// TwinCAT 3 PLC project SPS
// ProgramVersion: 3.1.4026.22
// libraries:
//   VisuElemMeter, * (System)
//   VisuElems, * (System)
//   VisuElemsSpecialControls, * (System)
//   VisuElemsWinControls, * (System)
//   VisuElemTextEditor, * (System)
//   VisuInputs, * (System)
//   VisuNativeControl, * (System)
//   Tc2_MC2, * (Beckhoff Automation GmbH)
//   Tc2_Standard, * (Beckhoff Automation GmbH)
//   Tc2_System, * (Beckhoff Automation GmbH)
//   Tc3_IotBase, * (Beckhoff Automation GmbH)
//   VisuSymbols, * (System)
// project tree:
//   GVLs/ GVL_PosKinematic.TcGVL, IFC_HW.TcGVL
//   / PlcTask.TcTTO
//   POUs/Abfüllmodul/ FB_Abfuellmodul.TcPOU, FB_Dispenser.TcPOU, FB_EZylinder.TcPOU, FB_Vereinzelung.TcPOU
//   POUs/ eBetriebszustand.TcDUT, FUN_Scale.TcPOU, MAIN.TcPOU
//   POUs/IoT/ FB_MQTT.TcPOU
//   POUs/Manipulator/ FB_Manipulator.TcPOU
//   POUs/Manipulator/Roboter/ FB_Roboter.TcPOU (not stored), FB_Roboter_Axis.TcPOU (not stored), FB_Roboter_E.TcPOU (not stored), FB_Roboter_Logik.TcPOU (not stored)
//   POUs/Statusleuchte/ FB_Ampelleuchte.TcPOU, FB_Blinklicht.TcPOU
// (motion and I/O tree: see PLC project lf_system_plc)
// real-time tasks:
//   TASK PlcTask: cycle T#10ms, priority 21, ADS port 350
//   TASK PlcTask1: cycle T#10ms, priority 22, ADS port 351
//   TASK PlcTask2: cycle T#10ms, priority 20, ADS port 352
//   TASK PlcTask3: cycle T#10ms, priority 23, ADS port 353
// variable links:

CONFIGURATION SPS
    RESOURCE PLC ON TwinCAT3
        TASK PlcTask(INTERVAL := T#10ms, PRIORITY := 23);
        PROGRAM MAIN WITH PlcTask : MAIN;
    END_RESOURCE
END_CONFIGURATION

// ---- POUs/eBetriebszustand.TcDUT
{attribute 'qualified_only'}
{attribute 'strict'}
{attribute 'to_string'}
TYPE eBetriebszustand :
(
	Off        := 0,   // nicht betriebsbereit
	Error      := 1,   // Fehlerbehafteter Stop
	Setup      := 2,   // Wartung
	Warning    := 3,   // nicht fehlerbehafteter, nicht geplanter Stop
	Init       := 4,   // Herstellung Betriebsbereitschaft
	Ready      := 5,   // betriebsbereit
	Production := 6,   // Betrieb
	Done       := 7,   // Betrieb abgeschlossen
	Stop       := 8
);
END_TYPE

// ---- GVLs/GVL_PosKinematic.TcGVL
{attribute 'qualified_only'}
VAR_GLOBAL
	// Home position
	pXhome : REAL := 29;
	pYhome : REAL := 145.5;
	pZhome : REAL := 45;
	
	// Conveyor position
	pXconv : REAL := 29;
	pYconv : REAL := 145.5;
	pZconv : REAL := 130;
	
	//Scale position
	pXscale : REAL := 36;
	pYscale : REAL := 7.5;
	pZscale : REAL := 131.5;
	
	// Heating position
	pXheat : REAL := 218.5;
	pYheat : REAL := 7;
	pZheat : REAL := 159;
	
	// Storage position
	pX1stor : REAL := 107;
	pX2stor : REAL := 158.7;
	pX3stor : REAL := 209.3;
	pX4stor : REAL := 260.3;
	pYstor : REAL := 139;
	pZstor : REAL := 120;
	
	// Z offset height
	pZoff : REAL := 45;
END_VAR

// ---- GVLs/IFC_HW.TcGVL
// In dieser GVL werden alle Variablen deklariert die auf die realen Klemmen zugreifen
VAR_GLOBAL
	
	// Allgemeine Variablen fur MAIN und HMI
		bEnable		AT%I*	: BOOL;			// Enable Factory (HMI Production Umgebung)
		bExecute	AT%I*	: BOOL;			// Startsignal	(Start Knopf Konsole)
		bStop				: BOOL;			// Stop Variable (interne Variable um FB's zu stoppen)
		
	// Station Statusampel	
		bAmpelRot 	AT%Q* 	: BOOL;			// Signal-LED Rot
		bAmpelGelb 	AT%Q* 	: BOOL;			// Signal-LED Gelb
		bAmpelGrun 	AT%Q* 	: BOOL;			// Signal-LED Grun
			
	// Station Vereinzelung
		bEinzelSens1 	AT%I*	: BOOL;					// Separation Sensor 1 (Kammer)
		bEinzelSens2 	AT%I*	: BOOL;					// Separation Sensor 2 (Rohr)
		bEinzelSens3 	AT%I*	: BOOL;					// Separation Sensor 3 (Flasche auf Kopf)
		bR1AKT1 		AT%Q* 	: BOOL := FALSE;		// Relais 1 Aktor 1 (Schleuse Oben öffnen)
		bR2AKT1 		AT%Q* 	: BOOL := TRUE; 		// Relais 2 Aktor 1 (Schleuse Oben schließen)
		bR1AKT2 		AT%Q* 	: BOOL := FALSE;		// Relais 1 Aktor 2 (Schleuse Unten öffne)
		bR2AKT2 		AT%Q* 	: BOOL := TRUE;			// Relais 2 Aktor 2	(Schleuse Unten schließen)
	
	// Station Forderband
		bBandSens1 	AT %I*	: BOOL;		// Forderband Sensor 1 (Extruder 1)
		bBandSens2	AT %I*	: BOOL;		// Forderband Sensor 2 (Extruder 2)
		bBandSens3 	AT %I*	: BOOL;		// Forderband Sensor 3 (Extruder 3)
		bBandSens4 	AT %I*	: BOOL;		// Forderband Sensor 4 (Übergabe Roboter)
		bBandHub1 	AT %Q*	: BOOL;		// Forderband Hubmagnet 1 (Schleuse Extruder 1)
		bBandHub2 	AT %Q*	: BOOL;		// Forderband Hubmagnet 1 (Schleuse Extruder 2)
		bBandHub3 	AT %Q*	: BOOL;		// Forderband Hubmagnet 1 (Schleuse Extruder 3)
		
		ax_Extruder1 	: AXIS_REF;		// Forderband NC-Achse Extruder 1
		ax_Extruder2 	: AXIS_REF;		// Forderband NC-Achse Extruder 2
		ax_Extruder3 	: AXIS_REF;		// Forderband NC-Achse Extruder 3
		ax_BandMotor 	: AXIS_REF;		// Forderband NC-Achse Band
		
		iBandFullmenge1		: INT := 1;	// in Gramm (Soll Füllmenge Extruder 1)
		iBandFullmenge2		: INT := 1;	// in Gramm (Soll Füllmenge Extruder 2)
		iBandFullmenge3		: INT := 1;	// in Gramm (Soll Füllmenge Extruder 3)
		
	//Füllstandsüberwachung
		iFillSens1 AT%I*	: UINT;		// Füllstandssensor im Granulatspeicher 1
		iFillSens2 AT%I*	: UINT;		// Füllstandssensor im Granulatspeicher 2
		iFillSens3 AT%I*	: UINT;		// Füllstandssensor im Granulatspeicher 3
		
		rFillLevelPercent1	: REAL;		// Füllstand im Granulatspeicher 1 in %
		rFillLevelGramm1	: REAL;		// Füllstand im Granulatspeicher 1 in g
		rFillLevelPercent2	: REAL;		// Füllstand im Granulatspeicher 2 in %
		rFillLevelGramm2	: REAL;		// Füllstand im Granulatspeicher 2 in g
		rFillLevelPercent3	: REAL;		// Füllstand im Granulatspeicher 3 in %
		rFillLevelGramm3	: REAL;		// Füllstand im Granulatspeicher 3 in g
		
		rMaxFillLevel 		: REAL := 375;	// Kalibrierter Füllstand für 10% * 10
		
	// Station Waage
		sWaageNachricht		: STRING;	// Nachricht von Wagezelle (fur virtuelle Inbetriebnahme notig)
		bWaageNull			: BOOL;		// TARA Waage (Waage auf Null setzen)
		iWaageMesswert		: INT;		// Messwert der Waage
		
	// Station Behalteridentifikation
		bIdSensorTrager		: BOOL;		// Sensor bei Erkennung eines Datentrager
		sIdNachricht		: STRING;	// Nachricht von RFID-System (fur virtuelle Inbetriebnahme notig)
		sSeriennummer		: STRING;	// Seriennummer RFID-Tag
		
	//Temperierstation
		bVentilator1 	AT %Q*	: BOOL;		// Ventilator 1
		bVentilator2 	AT %Q*	: BOOL;		// Ventilator 2
		bVentilator3 	AT %Q*	: BOOL;		// Ventilator 3
		
		iTempSens1 		AT%I*	: UINT;		// Temperatursensor 1
		iTempSens2 		AT%I*	: UINT;		// Temperatursensor 2
		iHeizpatrone 	AT%Q*	: UINT;		// Heizpatronen
		
		iMaxTemp				: UINT := 5500;		// in °C * 100
		
	// Station Manipulator
		bManEndXmin 		AT%I* 	: BOOL := TRUE;		// Manipulator min Endschalter Achse x
		bManEndYmin 		AT%I* 	: BOOL := TRUE;		// Manipulator min Endschalter Achse y
		bManEndZmin 		AT%I* 	: BOOL := TRUE;		// Manipulator min Endschalter Achse z
		bManEndGmin 		AT%I* 	: BOOL := TRUE;		// Manipulator min Endschalter Achse Gripper
		bManEndXmax 		AT%I* 	: BOOL := TRUE;		// Manipulator max Endschalter Achse x
		bManEndYmax 		AT%I* 	: BOOL := TRUE;		// Manipulator max Endschalter Achse y
		bManEndZmax 		AT%I* 	: BOOL := TRUE;		// Manipulator max Endschalter Achse z
		bManEndGmax 		AT%I* 	: BOOL := TRUE;		// Manipulator max Endschalter Achse Gripper
		bManBrakeZ			AT%Q*	: BOOL := FALSE;	// Bremse Achse z
		
		ax_ManX			: AXIS_REF;			// Manipulator NC-Achse x
		ax_ManY			: AXIS_REF;			// Manipulator NC-Achse y
		ax_ManZ			: AXIS_REF;			// Manipulator NC-Achse z
		ax_ManG			: AXIS_REF; 		// Manipulator NC-Achse Gripper
		
		bGripperClosed		AT%Q*	: BOOL; 			// signal if gripper is closed ONLY USED IN SIM
END_VAR

// ---- POUs/MAIN.TcPOU
PROGRAM MAIN
VAR
	fb_Ampelleuchte :FB_Ampelleuchte;	
	fb_Abfuellmodul :FB_Abfuellmodul;
	fb_Manipulator :FB_Manipulator;
	
	nState :INT :=0;
	
	fb_MQTT :FB_MQTT;
END_VAR

	
fb_Ampelleuchte(eState:= , bAmpelGruen_out=> IFC_HW.bAmpelGrun, bAmpelRot_out=> IFC_HW.bAmpelRot, bAmpelGelb_out=> IFC_HW.bAmpelGelb);

fb_Abfuellmodul(bEnable:= , bExecute:= , eState=> ); 
fb_Manipulator(bEnable:= , bExecute:= , bGripperClosed=> IFC_HW.bGripperClosed, eState=> );

IF fb_Abfuellmodul.eState = eBetriebszustand.Init OR fb_Manipulator.eState = eBetriebszustand.Init THEN
	fb_Ampelleuchte.eState := eBetriebszustand.init;
ELSIF fb_Abfuellmodul.eState = eBetriebszustand.ready AND fb_Manipulator.eState = eBetriebszustand.ready THEN
	fb_Ampelleuchte.eState := eBetriebszustand.ready;
ELSIF fb_Abfuellmodul.eState = eBetriebszustand.production OR fb_Manipulator.eState = eBetriebszustand.Production THEN
	fb_Ampelleuchte.eState := eBetriebszustand.Production;
ELSIF fb_Abfuellmodul.eState = eBetriebszustand.off AND fb_Manipulator.eState = eBetriebszustand.off THEN
	fb_Ampelleuchte.eState := eBetriebszustand.off;
ELSE 
	fb_Ampelleuchte.eState := eBetriebszustand.Warning;
END_IF


IF NOT IFC_HW.bEnable THEN
	nState :=0;
END_IF
CASE nState Of
	0://off
	fb_Abfuellmodul.bEnable :=FALSE;
	fb_Manipulator.bEnable :=FALSE;
	
	IF IFC_HW.bEnable THEN
		nstate:=1;
	END_IF
	
	1: //init
	fb_Abfuellmodul.bEnable :=TRUE;
	fb_Manipulator.bEnable :=TRUE;
	
	IF fb_Abfuellmodul.eState = eBetriebszustand.Ready AND fb_Manipulator.eState = eBetriebszustand.Ready THEN
		nState:=2;
	END_IF
	
	2: //ready
	IF IFC_HW.bExecute AND iFC_HW.bEinzelSens1 THEN
		nstate :=21;
	END_IF
	IF NOT iFC_HW.bEinzelSens2 AND NOT iFC_HW.bEinzelSens1 THEN
		fb_Abfuellmodul.bEnable :=FALSE;
		nState :=1;
	END_IF
	
	21: //bottle
	fb_Abfuellmodul.bExecute :=TRUE;
	
	IF fb_Abfuellmodul.eState = eBetriebszustand.Done THEN
		fb_Abfuellmodul.bExecute :=FALSE;
		nstate :=22;
	END_IF
	
	22: //mani
	fb_Manipulator.bExecute :=TRUE;
	
	IF fb_Manipulator.eState = eBetriebszustand.Done THEN
		fb_Manipulator.bExecute :=FALSE;
		nState :=23;
	END_IF
	
	23://done
	IF NOT IFC_HW.bExecute THEN
		nState:=2;
	END_IF
END_CASE


fb_MQTT(data:= IFC_HW.bEnable);

END_PROGRAM

// ---- POUs/Statusleuchte/FB_Ampelleuchte.TcPOU
FUNCTION_BLOCK FB_Ampelleuchte
VAR_INPUT
	eState : eBetriebszustand;
END_VAR
VAR_OUTPUT

	
	bAmpelGruen_out :BOOL;
	bAmpelRot_out :BOOL;
	bAmpelGelb_out :BOOL;
	
END_VAR
VAR
	fb_BlinklichtGr :FB_Blinklicht;
	fb_BlinklichtRt :FB_Blinklicht;
	fb_BlinklichtGb :FB_Blinklicht;
	AmpelGruenblinken:BOOL;
	AmpelRotblinken :BOOL;
	AmpelGelbblinken :BOOL;
	bAmpelGruen :BOOL;
	bAmpelRot :BOOL;
	bAmpelGelb :BOOL;
END_VAR

CASE eState OF
	0: //OFF nicht Betriebsbereit
	//keine Lampe leuchtet
	bAmpelGruen :=FALSE;
	bAmpelRot :=FALSE;
	bAmpelGelb :=FALSE;
	AmpelGruenblinken:=FALSE;
	AmpelRotblinken :=FALSE;
	AmpelGelbblinken :=FALSE;
	
	1: //Error Fehlerbehafteter Stop (Sicherheitssteuerung)
	//Rote Lampe Leuchtet 
	bAmpelGruen :=FALSE;
	bAmpelRot :=TRUE;
	bAmpelGelb :=FALSE;
	AmpelGruenblinken:=FALSE;
	AmpelRotblinken :=FALSE;
	AmpelGelbblinken :=FALSE;
	
	2: //Setup Wartung
	//Rot und Gelb blinkt
	bAmpelGruen :=FALSE;
	bAmpelRot :=FALSE;
	bAmpelGelb :=FALSE;
	AmpelGruenblinken:=FALSE;
	AmpelRotblinken :=TRUE;
	AmpelGelbblinken :=TRUE;
	
	3: //Warning Nicht Fehlerbehafteter nicht geplanter Stop
	//Gelb blinken
	bAmpelGruen :=FALSE;
	bAmpelRot :=FALSE;
	bAmpelGelb :=FALSE;
	AmpelGruenblinken:=FALSE;
	AmpelRotblinken :=FALSE;
	AmpelGelbblinken :=TRUE;
	
	4: //Init Herstellung Betriebsbereitschaft
	//Gelb Grün blinkt
	bAmpelGruen :=FALSE;
	bAmpelRot :=FALSE;
	bAmpelGelb :=FALSE;
	AmpelGruenblinken:=TRUE;
	AmpelRotblinken :=FALSE;
	AmpelGelbblinken :=TRUE;
	
	5: //Ready Betriebsbereit
	//Grün blinkt
	bAmpelGruen :=FALSE;
	bAmpelRot :=FALSE;
	bAmpelGelb :=FALSE;
	AmpelGruenblinken:=TRUE;
	AmpelRotblinken :=FALSE;
	AmpelGelbblinken :=FALSE;
	
	6: //Production Betrieb
	//Grün leuchtet
	bAmpelGruen :=TRUE;
	bAmpelRot :=FALSE;
	bAmpelGelb :=FALSE;
	AmpelGruenblinken:=FALSE;
	AmpelRotblinken :=FALSE;
	AmpelGelbblinken :=FALSE;
	
	7: //Done Betrieb abgeschlossen 
	//Grün Gelb leuchten
	bAmpelGruen :=TRUE;
	bAmpelRot :=FALSE;
	bAmpelGelb :=TRUE;
	AmpelGruenblinken:=FALSE;
	AmpelRotblinken :=FALSE;
	AmpelGelbblinken :=FALSE;
	
	8: //Stop
	//Rot blinken
	bAmpelGruen :=FALSE;
	bAmpelRot :=FALSE;
	bAmpelGelb :=FALSE;
	AmpelGruenblinken:=FALSE;
	AmpelRotblinken :=TRUE;
	AmpelGelbblinken :=FALSE;
END_CASE

fb_BlinklichtGb(bStartStop:= AmpelGelbblinken, tPeriod:= T#1S , bBlink=> );
fb_BlinklichtGr(bStartStop:= AmpelGruenblinken, tPeriod:= T#1S, bBlink=> );
fb_BlinklichtRt(bStartStop:= AmpelRotblinken, tPeriod:= T#1S, bBlink=> );

IF fb_BlinklichtGb.bBlink OR bAmpelGelb THEN
	bAmpelGelb_out :=TRUE;
ELSE
	bAmpelGelb_out :=FALSE;
END_IF
IF fb_BlinklichtGr.bBlink OR bAmpelGruen THEN
	bAmpelGruen_out :=TRUE;
ELSE
	bAmpelGruen_out :=FALSE;
END_IF
IF fb_BlinklichtRt.bBlink OR bAmpelRot THEN
	bAmpelRot_out :=TRUE;
ELSE
	bAmpelRot_out :=FALSE;
END_IF

END_FUNCTION_BLOCK

// ---- POUs/Statusleuchte/FB_Blinklicht.TcPOU
FUNCTION_BLOCK FB_Blinklicht
VAR_INPUT
	bStartStop :BOOL;
	tPeriod :TIME := T#1s;
	
END_VAR
VAR_OUTPUT
	bBlink :BOOL;
	
END_VAR
VAR
	fbTON :TON;
	fbRtrig :R_Trig;
	bEinAus :BOOL := 0;
END_VAR

fbRtrig(CLK:= bStartStop, Q=> );

IF fbRtrig.Q THEN
	bEinAus:= NOT bEinAus;
END_IF


//fbTON.IN := bBlink AND NOT fbTON.Q;
//fbTON.PT:=T#1S;

fbTON(in:=bEinAus AND NOT fbTON.Q , PT:= tPeriod, Q=>,ET=>);

IF fbTON.ET<=fbTON.PT/2 THEN
	bBlink := FALSE;
ELSIF fbTON.ET>fbTON.PT/2 THEN
	bBlink := TRUE;
END_IF

(*IF NOT bBlink THEN
	bLEDrot := FALSE;
END_IF
*)

IF NOT bStartStop THEN
	bBlink :=FALSE;
END_IF

END_FUNCTION_BLOCK

// ---- POUs/Abfüllmodul/FB_Abfuellmodul.TcPOU
FUNCTION_BLOCK FB_Abfuellmodul
VAR_INPUT
	bEnable :BOOL;
	bExecute :BOOL;
END_VAR
VAR_OUTPUT
	eState :eBetriebszustand;
END_VAR
VAR
	fb_Vereinzelung :FB_Vereinzelung;
	fb_Transport : FB_Transport;
	fb_Dispenser1 :FB_Dispenser;
	fb_Dispenser2 :FB_Dispenser;
	fb_Dispenser3 :FB_Dispenser;
	fb_EZylinder1 : FB_EZylinder;
	fb_EZylinder2 : FB_EZylinder;

	
	nState :INT;
	nStation :INT;
END_VAR

fb_Vereinzelung(
	bEnable:= , 
	bExecute:= , 
	bSens1:= IFC_HW.bEinzelSens1, 
	bSens2:= IFC_HW.bEinzelSens2, 
	bSens3:= IFC_HW.bEinzelSens3, 
	bSens4:= IFC_HW.bBandSens1, 
	eState=> , 
	bGate1=> fb_EZylinder1.bGate, 
	bGate2=> fb_EZylinder2.bGate);
	
fb_Transport(
	bEnable:= , 
	bExecute:= , 
	nStation:= nStation, 
	bSens1:= IFC_HW.bBandSens1, 
	bSens2:= IFC_HW.bBandSens2, 
	bSens3:= IFC_HW.bBandSens3, 
	bSens4:= IFC_HW.bBandSens4, 
	eState=> , 
	bStopper1=> IFC_HW.bBandHub1, 
	bStopper2=> IFC_HW.bBandHub2, 
	bStopper3=> IFC_HW.bBandHub3, 
	ax:= IFC_HW.ax_BandMotor);
	
fb_Dispenser1(
	bEnable:= , 
	bExecute:= , 
	rDistance:= IFC_HW.iBandFullmenge1*20, 
	eState=> , 
	ax:= IFC_HW.ax_Extruder1);
fb_Dispenser2(
	bEnable:= , 
	bExecute:= , 
	rDistance:= IFC_HW.iBandFullmenge1*20, 
	eState=> , 
	ax:= IFC_HW.ax_Extruder2);
fb_Dispenser3(
	bEnable:= , 
	bExecute:= , 
	rDistance:= IFC_HW.iBandFullmenge1*20, 
	eState=> , 
	ax:= IFC_HW.ax_Extruder3);
	
fb_EZylinder1(bGate:= , bError:= , bR1=> IFC_HW.bR1AKT1, bR2=> IFC_HW.bR2AKT1);
fb_EZylinder2(bGate:= , bError:= , bR1=> IFC_HW.bR1AKT2, bR2=> IFC_HW.bR2AKT2);


IF NOT bEnable THEN 
	nState :=0;
END_IF


CASE nState OF
	0: // Off
	eState := eBetriebszustand.Off;
	
	fb_Vereinzelung.bEnable:=FALSE;
	fb_Transport.bEnable :=FALSE;
	fb_Dispenser1.bEnable :=FALSE;
	fb_Dispenser2.bEnable :=FALSE;
	fb_Dispenser3.bEnable :=FALSE;
	fb_Vereinzelung.bExecute :=FALSE;
	fb_Transport.bExecute :=FALSE;
	fb_Dispenser1.bExecute :=FALSE;
	fb_Dispenser2.bExecute :=FALSE;
	fb_Dispenser3.bExecute :=FALSE;
	
	IF bEnable THEN
		nstate :=10;
	END_IF
	
	10:// Init
	eState := eBetriebszustand.Init;
	
	fb_Vereinzelung.bEnable:=TRUE;
	fb_Transport.bEnable :=TRUE;
	fb_Dispenser1.bEnable :=TRUE;
	fb_Dispenser2.bEnable :=TRUE;
	fb_Dispenser3.bEnable :=TRUE;
	fb_Vereinzelung.bExecute :=FALSE;
	fb_Transport.bExecute :=FALSE;
	fb_Dispenser1.bExecute :=FALSE;
	fb_Dispenser2.bExecute :=FALSE;
	fb_Dispenser3.bExecute :=FALSE;
	
	IF (fb_Vereinzelung.eState = eBetriebszustand.Ready) AND (fb_Transport.eState = eBetriebszustand.Ready) AND (fb_Dispenser1.eState = eBetriebszustand.Ready) AND (fb_Dispenser2.eState = eBetriebszustand.Ready) AND (fb_Dispenser3.eState = eBetriebszustand.Ready)THEN
		nstate :=20;
	END_IF
	
	20:// Ready
	eState := eBetriebszustand.Ready;
	
	fb_Vereinzelung.bEnable:=TRUE;
	fb_Transport.bEnable :=TRUE;
	fb_Dispenser1.bEnable :=TRUE;
	fb_Dispenser2.bEnable :=TRUE;
	fb_Dispenser3.bEnable :=TRUE;
	fb_Vereinzelung.bExecute :=FALSE;
	fb_Transport.bExecute :=FALSE;
	fb_Dispenser1.bExecute :=FALSE;
	fb_Dispenser2.bExecute :=FALSE;
	fb_Dispenser3.bExecute :=FALSE;
	
	IF bExecute THEN
		nState:=30;
	END_IF
	
	30:// Start
	eState := eBetriebszustand.Production;
	
	fb_Vereinzelung.bExecute :=TRUE;
	fb_Transport.bExecute :=TRUE;
	fb_Dispenser1.bExecute :=FALSE;
	fb_Dispenser2.bExecute :=FALSE;
	fb_Dispenser3.bExecute :=FALSE;
	nStation :=1;
	
	IF (fb_Vereinzelung.eState = eBetriebszustand.Done) AND (fb_Transport.eState = eBetriebszustand.Done) THEN
		nstate :=31;
	END_IF
	
	31:// Dispenser1
	eState := eBetriebszustand.Production;
	
	fb_Vereinzelung.bExecute :=FALSE;
	fb_Transport.bExecute :=FALSE;
	fb_Dispenser1.bExecute :=TRUE;
	fb_Dispenser2.bExecute :=FALSE;
	fb_Dispenser3.bExecute :=FALSE;
	nStation :=1;
	
	IF fb_Dispenser1.eState = eBetriebszustand.Done THEN
		nState :=32;
	END_IF
	
	32:// Bewegung zu Dispenser2
	eState := eBetriebszustand.Production;
	
	nStation :=2;
	fb_Vereinzelung.bExecute :=FALSE;
	fb_Transport.bExecute :=TRUE;
	fb_Dispenser1.bExecute :=FALSE;
	fb_Dispenser2.bExecute :=FALSE;
	fb_Dispenser3.bExecute :=FALSE;
	
	IF fb_Transport.eState = eBetriebszustand.Done THEN
		nState :=33;
	END_IF
	
	33:// Dispenser2
	eState := eBetriebszustand.Production;
	
	fb_Vereinzelung.bExecute :=FALSE;
	fb_Transport.bExecute :=FALSE;
	fb_Dispenser1.bExecute :=FALSE;
	fb_Dispenser2.bExecute :=TRUE;
	fb_Dispenser3.bExecute :=FALSE;
	nStation :=2;
	
	IF fb_Dispenser2.eState = eBetriebszustand.Done THEN
		nState :=34;
	END_IF
		
	34:// Bewegung zu Dispenser3
	eState := eBetriebszustand.Production;
	
	nStation :=3;
	fb_Vereinzelung.bExecute :=FALSE;
	fb_Transport.bExecute :=TRUE;
	fb_Dispenser1.bExecute :=FALSE;
	fb_Dispenser2.bExecute :=FALSE;
	fb_Dispenser3.bExecute :=FALSE;
	
	IF fb_Transport.eState = eBetriebszustand.Done THEN
		nState :=35;
	END_IF
	
	35:// Dispenser3
	eState := eBetriebszustand.Production;
	
	fb_Vereinzelung.bExecute :=FALSE;
	fb_Transport.bExecute :=FALSE;
	fb_Dispenser1.bExecute :=FALSE;
	fb_Dispenser2.bExecute :=FALSE;
	fb_Dispenser3.bExecute :=TRUE;
	nStation :=3;
	
	IF fb_Dispenser3.eState = eBetriebszustand.Done THEN
		nState :=36;
	END_IF
	
	36:// Abholstation
	eState := eBetriebszustand.Production;
	
	nStation :=4;
	fb_Vereinzelung.bExecute :=FALSE;
	fb_Transport.bExecute :=TRUE;
	fb_Dispenser1.bExecute :=FALSE;
	fb_Dispenser2.bExecute :=FALSE;
	fb_Dispenser3.bExecute :=FALSE;
		
	IF fb_Transport.eState = eBetriebszustand.Done THEN
		nState :=40;
	END_IF 
	
	40:// Done
	eState := eBetriebszustand.Done;
	
	fb_Vereinzelung.bExecute :=FALSE;
	fb_Transport.bExecute :=FALSE;
	fb_Dispenser1.bExecute :=FALSE;
	fb_Dispenser2.bExecute :=FALSE;
	fb_Dispenser3.bExecute :=FALSE;
	
	IF not bExecute THEN
		nState :=20;
	END_IF
	
	
END_CASE

END_FUNCTION_BLOCK

// ---- POUs/Abfüllmodul/FB_Vereinzelung.TcPOU
FUNCTION_BLOCK FB_Vereinzelung
VAR_INPUT
	//Steuervariablen
	bEnable :BOOL;
	bExecute :BOOL;
	
	//Hardwareeingänge
	bSens1 :BOOL; //Flasche in der Kammer
	bSens2 :BOOL; //Flasche im Rohr
	bSens3 :BOOL; //Flasche verkehrt
	bSens4 :BOOL; //Flasche am Förderband
END_VAR
VAR_OUTPUT
	//Steuervariable 
	eState :eBetriebszustand;
	
	//Hardwareausgägne
	bGate1 :BOOL;
	bGate2 :BOOL;
END_VAR
VAR
	nState :INT :=100;
	fbTON :TON;
END_VAR

fbTON(IN:= , PT:= T#2S, Q=> , ET=> );

IF NOT bEnable THEN
	nState :=0;
END_IF

CASE nState OF
	100: //Off oder nicht Betriebsbereit 
	eState:=eBetriebszustand.Off;
	
	IF bSens1 AND bEnable THEN
		nState:=21; //Ready
	ELSIF bEnable THEN
		nState :=0; //Init
	END_IF
	
	
	0: //Kammer ist leer
	eState:=eBetriebszustand.Init;
	
	bGate1:=FALSE;
	bGate2:=FALSE;
	
	IF bSens2 THEN
		nState:=1; //Oben öffnen
	END_IF
	
	
	1: //Oben öffnen
	eState := eBetriebszustand.Init;
	
	bGate1:=TRUE;
	bGate2 :=FALSE;
	
	IF bSens1 THEN
		nState:=2; //Oben schleißen
	END_IF
	
	
	2: //Oben schließen
	eState := eBetriebszustand.Init;
	
	bGate1:=FALSE;
	bGate2 :=FALSE;
	fbTon.IN:=TRUE;
	
	IF fbTon.Q THEN
		nState:=21; //Ready
		fbTon.IN :=FALSE;
	END_IF
	
	21: //Ready
	eState := eBetriebszustand.Ready;
	
	bGate1:=FALSE;
	bGate2 :=FALSE;
	
	IF bExecute THEN
		nState:=3; //Unten öffnen
	END_IF
	
	
	3: //Unten öffnen
	eState := eBetriebszustand.Production;
	
	bGate1:=FALSE;
	bGate2 :=TRUE;
	
	IF bSens4 THEN
		nState :=4; //Unten schließen
	END_IF
	
	4: //Unten schließen
	eState := eBetriebszustand.Production;
	
	bGate1:=FALSE;
	bGate2 :=FALSE;
	fbTon.IN :=TRUE;
	
	IF fbTon.Q THEN
		nState:=41; //Done
		fbTon.IN :=FALSE;
	END_IF
	
	41: //Done
	eState:= eBetriebszustand.Done;
	
	IF NOT bExecute THEN
		nState :=0; //Kammer leer
	END_IF
	
	
END_CASE

END_FUNCTION_BLOCK

// ---- POUs/Abfüllmodul/FB_Dispenser.TcPOU
FUNCTION_BLOCK FB_Dispenser
VAR_INPUT
	bEnable :BOOL;
	bExecute :BOOL;
	rDistance :REAL;
END_VAR
VAR_OUTPUT
	eState :eBetriebszustand;
END_VAR
VAR
	mc_Reset :MC_Reset;
	mc_Power :MC_Power;
	mc_MoveRelative :MC_MoveRelative;
	nState :INT :=0;
END_VAR
VAR_IN_OUT
	ax :Axis_Ref;
END_VAR

ax.ReadStatus();
mc_Reset(
	Axis:= ax, 
	Execute:= , 
	Done=> , 
	Busy=> , 
	Error=> , 
	ErrorID=> );
	
mc_Power(
	Axis:= ax, 
	Enable:= , 
	Enable_Positive:= , 
	Enable_Negative:= , 
	Override:= , 
	BufferMode:= , 
	Options:= , 
	Status=> , 
	Busy=> , 
	Error=> , 
	ErrorID=> );
	
mc_MoveRelative(
	Axis:= ax, 
	Execute:= , 
	Distance:= rDistance, 
	Velocity:= 60, 
	Acceleration:= 30, 
	Deceleration:= 30, 
	Jerk:= , 
	BufferMode:= , 
	Options:= , 
	Done=> , 
	Busy=> , 
	Active=> , 
	CommandAborted=> , 
	Error=> , 
	ErrorID=> );
	

IF NOT bEnable THEN
	nState:=0;
END_IF

CASE nState OF 
	0:
	eState:=eBetriebszustand.Off;
	mc_Power.Enable :=TRUE;
	mc_Power.Enable_Positive:=TRUE;
	
	
	IF bEnable AND NOT mc_power.Status THEN
		nState :=10;
	ELSIF mc_power.Status AND bEnable THEN
		nState:=20;
	END_IF
	
	10: // init Reset
	eState:=eBetriebszustand.Init;
	mc_Reset.Execute:=TRUE;
	
	IF mc_Reset.Done THEN
		nState:=11;
	END_IF
	
	11: // init Power
	eState:=eBetriebszustand.Init;
	mc_Reset.Execute:=FALSE;
	mc_Power.Enable :=TRUE;
	mc_Power.Enable_Positive:=TRUE;
	
	
	IF mc_Power.Status THEN
		nState:=20;
	END_IF
	
	20: // Ready
	eState:= eBetriebszustand.Ready;
	
	IF bExecute THEN 
		nState:=30;
	END_IF
 
	30: // Kontinuierliche Bewegung
	eState:=eBetriebszustand.Production;
	mc_MoveRelative.Execute :=TRUE;
	
	IF mc_MoveRelative.Done THEN 
		mc_MoveRelative.Execute:=FALSE;
		nState :=40;
	END_IF
	
	40: // Fertig
	eState :=eBetriebszustand.Done;
	
	IF NOT bExecute THEN 
		nState:=20;
	END_IF

END_CASE

END_FUNCTION_BLOCK

// ---- POUs/Abfüllmodul/FB_EZylinder.TcPOU
FUNCTION_BLOCK FB_EZylinder
VAR_INPUT
	bGate :BOOL;
	bError :BOOL;
END_VAR
VAR_OUTPUT
	bR1 :BOOL;
	bR2 :BOOL;
END_VAR
VAR
END_VAR

bR1 :=bGate;
bR2 := NOT bGate;

IF bError THEN
	bR1 := FALSE;
	bR2 := FALSE;
END_IF

END_FUNCTION_BLOCK

// ---- POUs/Manipulator/FB_Manipulator.TcPOU
FUNCTION_BLOCK FB_Manipulator
VAR_INPUT
	bEnable :BOOL; 
	bExecute :BOOL; //Sensor band 
END_VAR
VAR_OUTPUT
	bGripperClosed :BOOL;
	eState :eBetriebszustand;
END_VAR
VAR
	fb_Roboter :FB_Roboter;
	fb_Roboter_Gripper : FB_Roboter_Axis;
	fb_Gripper_E :FB_Roboter_E;
	//FB_waage
	//FB temp
	
	
	nState :INT :=0;
	nStation :INT :=0; 
	pPositionX :REAL;
	pPositionY :REAL;
	pPositionZ :REAL;
	
	
	
	
	nBottles: INT :=0;
END_VAR

fb_Roboter(
	bEnable:= , 
	bExecute:= , 
	pPositionX:= pPositionX, 
	pPositionY:= pPositionY, 
	pPositionZ:= pPositionZ, 
	eState=> );
	
fb_Gripper_E(bRefMax_in:= bManEndGmax, bRefMin_in:= bManEndGmin, bRefMax_out=> , bRefMin_out=> );
fb_Roboter_Gripper(
	bEnable:= , 
	bExecute:= , 
	rPosition:= , 
	bRefSens:= fb_Gripper_E.bRefMin_out, 
	eState=> , 
	ax:= IFC_HW.ax_ManG);
	
IF NOT bEnable THEN
	nState :=0;
END_IF	
	
	
CASE nState OF 
	0: //off
	eState:=eBetriebszustand.Off;
	IF bEnable THEN
		nState:=1;
	END_IF
	
	1: //init
	eState:=eBetriebszustand.Init;
	nbottles :=0;
	fb_Roboter_Gripper.bEnable:=TRUE;
	fb_Roboter.bEnable :=TRUE;
	
	IF (fb_Roboter_Gripper.eState = eBetriebszustand.Ready) AND (fb_Roboter.eState = eBetriebszustand.Ready) THEN 
		nState:=2;
	END_IF
	
	2://home 
	eState:=eBetriebszustand.Init;
	nStation :=0;
	fb_Roboter.bExecute :=TRUE;
	fb_Roboter_Gripper.rPosition := 7; //offen;
	fb_Roboter_Gripper.bExecute :=TRUE;
	bGripperClosed :=FALSE;
	
	IF (fb_Roboter_Gripper.eState = eBetriebszustand.Done) AND (fb_Roboter.eState = eBetriebszustand.Done) THEN 
		fb_Roboter.bExecute :=FALSE;
		fb_Roboter_Gripper.bExecute :=FALSE;
		nState:=20;
	END_IF
	
	20: //Ready
	IF nstation =7 THEN
		eState:=eBetriebszustand.Stop;
		//zusätzlicher State  bei dem man nur mit quittierung rauskommt 
	ELSE
			eState:=eBetriebszustand.Ready;
	END_IF
	
	nStation :=0;
	
	IF bExecute THEN 
		nState:=21;
	END_IF
	
	21: //open gripper
	eState:=eBetriebszustand.Production;
	fb_Roboter_Gripper.rPosition := 7; //offen;
	fb_Roboter_Gripper.bExecute :=TRUE;
	bGripperClosed :=FALSE;
	
	IF fb_Roboter_Gripper.eState = eBetriebszustand.Done THEN 
		fb_Roboter_Gripper.bExecute :=FALSE;
		nState:=22;
		
	END_IF
	
	22: //move to position
	eState:= eBetriebszustand.Production;
	nstation := 1;
	fb_Roboter.bExecute :=TRUE;
	
	IF fb_Roboter.eState = eBetriebszustand.Done THEN
		fb_Roboter.bExecute :=FALSE;
		nstate:=23;
	END_IF
	
	23: //close Gripper
	eState:=eBetriebszustand.Production;
	fb_Roboter_Gripper.rPosition := 9.4; //geschlossen;
	fb_Roboter_Gripper.bExecute :=TRUE;
	bGripperClosed :=TRUE;
	
	IF fb_Roboter_Gripper.eState = eBetriebszustand.Done THEN 
		fb_Roboter_Gripper.bExecute :=FALSE;
		nState:=24;
		nstation := nStation+1;
	END_IF
	
	24://move to new position
	eState:= eBetriebszustand.Production;
	
	fb_Roboter.bExecute :=TRUE;
	
	IF fb_Roboter.eState = eBetriebszustand.Done THEN
		fb_Roboter.bExecute :=FALSE;
		nstate:=25;
	END_IF
	
	25: //open gripper
	eState:=eBetriebszustand.Production;
	fb_Roboter_Gripper.rPosition := 7; //offen;
	fb_Roboter_Gripper.bExecute :=TRUE;
	bGripperClosed :=FALSE;
	
	IF fb_Roboter_Gripper.eState = eBetriebszustand.Done THEN 
		fb_Roboter_Gripper.bExecute :=FALSE;
		nState:=26;
	END_IF
	
	26: //do Position
	eState:=eBetriebszustand.Production;
	IF nStation >3 THEN
		nbottles := nBottles +1;
		nstate :=27;
	ELSIF nStation =3 THEN
		//wait
		nStation:= nstation +nBottles;
		nstate :=23;
	ELSIF nstation =2 THEN
		//wait
		nstate :=23;
	ELSE 
		nstate :=23;
	END_IF
	
	27: //Done
	eState:=eBetriebszustand.Done;
	IF NOT bExecute THEN 
		nstate:=2;
	END_IF
END_CASE



CASE nStation OF
	0: //Home
	pPositionX :=GVL_PosKinematic.pXhome;
	pPositionY :=GVL_PosKinematic.pYhome;
	pPositionZ :=GVL_PosKinematic.pZhome;
	//fb home
	
	1: //Conveyor
	pPositionX :=GVL_PosKinematic.pXconv;
	pPositionY :=GVL_PosKinematic.pYconv;
	pPositionZ:=GVL_PosKinematic.pZconv;
	//Fbconvoyer
	
	2: //Scale
	pPositionX :=GVL_PosKinematic.pXscale;
	pPositionY :=GVL_PosKinematic.pYscale;
	pPositionZ:=GVL_PosKinematic.pZscale;
	//scale wait
	
	3: //Heating
	pPositionX :=GVL_PosKinematic.pXheat;
	pPositionY :=GVL_PosKinematic.pYheat;
	pPositionZ:=GVL_PosKinematic.pZheat;
	//fb heating
	
	4: //storage1
	pPositionX :=GVL_PosKinematic.pX1stor;
	pPositionY :=GVL_PosKinematic.pYstor;
	pPositionZ:=GVL_PosKinematic.pZstor;
	
	5: //storage2
	pPositionX :=GVL_PosKinematic.pX2stor;
	pPositionY :=GVL_PosKinematic.pYstor;
	pPositionZ:=GVL_PosKinematic.pZstor;
	
	6: //storage3
	pPositionX :=GVL_PosKinematic.pX3stor;
	pPositionY :=GVL_PosKinematic.pYstor;
	pPositionZ:=GVL_PosKinematic.pZstor;
	
	7: //storage4
	pPositionX :=GVL_PosKinematic.pX4stor;
	pPositionY :=GVL_PosKinematic.pYstor;
	pPositionZ:=GVL_PosKinematic.pZstor;
	
	
END_CASE

END_FUNCTION_BLOCK

// ---- POUs/IoT/FB_MQTT.TcPOU
FUNCTION_BLOCK FB_MQTT
VAR
    fbMqttClient: FB_IotMqttClient; // MQTT client with initialization
    sTopicToPublish: STRING(255) := '$$groupsname: Die3Muskebiere'; // MQTT topic for temperature
	sMessageToPublish: STRING(255); // Message buffer
    tmrSendMessageInterval: TON := (PT := T#10S); // Interval timer for publishing
	nstate :int :=0;
END_VAR
VAR_INPUT
	data :BOOL;
END_VAR




CASE nstate OF 
	0:
		fbMqttClient.sHostName := '158.180.44.197';
		fbMqttClient.nHostPort := 1883;
		fbMqttClient.sTopicPrefix := 'aut/Die3Muskebiere';
		fbMqttClient.sClientId := 'Publishing PLC';
		fbMqttClient.sUserName := 'bobm';
		fbMqttClient.sUserPassword := 'letmein';
		fbMqttClient.Execute(bConnect := TRUE);
		IF fbMqttClient.bConnected THEN
			nstate :=1;
		END_IF
	
	1: 
		sMessageToPublish :='Die3Muskebiere';	
		fbMqttClient.Publish(
			sTopic := '/$$groupsname',
			pPayload := ADR('Die3Muskebiere'),
			nPayloadSize := LEN(sMessageToPublish) + 1,
			eQoS := TcIotMqttQos.AtMostOnceDelivery,
			bRetain := TRUE,
			bQueue := FALSE
		);
		nstate :=2;
	2:
		sMessageToPublish :='Oberhofer-Schrott-Hofer';	
		fbMqttClient.Publish(
			sTopic := '/name',
			pPayload := ADR(sMessageToPublish),
			nPayloadSize := LEN(sMessageToPublish) + 1,
			eQoS := TcIotMqttQos.AtMostOnceDelivery,
			bRetain := TRUE,
			bQueue := FALSE
		);
		nstate:=3;
	3:
		tmrSendMessageInterval(IN :=TRUE);
		IF tmrSendMessageInterval.Q THEN
			tmrSendMessageInterval(IN := FALSE);
			sMessageToPublish := BOOL_TO_STRING(data);
	
			fbMqttClient.Publish(
				sTopic := '/bEnable',
				pPayload := ADR(sMessageToPublish),
				nPayloadSize := LEN(sMessageToPublish) + 1,
				eQoS := TcIotMqttQos.AtMostOnceDelivery,
				bRetain := TRUE,
				bQueue := FALSE
			);
			fbMqttClient.Publish(
				sTopic := '/bEnable/$$unit',
				pPayload := ADR('bool'),
				nPayloadSize := LEN(sMessageToPublish) + 1,
				eQoS := TcIotMqttQos.AtMostOnceDelivery,
				bRetain := TRUE,
				bQueue := FALSE
			);
		END_IF
	
	
END_CASE

END_FUNCTION_BLOCK

// ---- POUs/FUN_Scale.TcPOU
FUNCTION FUN_Scale : REAL
VAR_INPUT
	ix :UINT;
	ix_max :REAL;
	ix_min :REAL;
	ry_min :REAL;
	ry_max :REAL;
END_VAR
VAR
	rk :REAL :=0.0854492188; //für Dispenser Ultraschallsensor 
	rd :REAL :=0;
END_VAR

//FUN keine deklarierung im Hauptprogramm

rk:=(ry_max-ry_min)/(ix_max-ix_min);
rd:=ry_min-rk*ix_min;

FUN_Scale := rk*ix+rd;

IF FUN_Scale > ry_max THEN
	FUN_Scale:=ry_max;
ELSIF FUN_Scale < ry_min THEN
	FUN_Scale:=ry_min;
END_IF

END_FUNCTION
